PROGRAM MAIN
VAR
END_VAR

END_PROGRAM

(* stored: Version 1.1.0.1
   POU MAIN: Id {adbb4842-6b2c-4856-8c9e-717ccd30de18} *)
